// TIA Portal V19 export
DATA_BLOCK "Com_FromPolygonFiller"   // DB471
{ S7_Optimized_Access := 'TRUE' }
// stored: AutoNumber false, MemoryReserve 0
   VAR RETAIN
      CIP : Struct   // CIP Signals From Hassia
         LifeBit : Bool;   // Watchdog bit
         RequestCIPLye : Bool;   // Request Lye Only CIP
         RequestCIPLyeAcid : Bool;   // Request Lye + Acid CIP
         SpareBool_0_3 : Bool;
         SpareBool_0_4 : Bool;
         SpareBool_0_5 : Bool;
         SpareBool_0_6 : Bool;
         SpareBool_0_7 : Bool;
         CIPRunning : Bool;
         NoTimeStop : Bool;
         ReleaseCIPFeedPump : Bool;
         CipReturnPumpRunning : Bool;
         RequestPreRinse_1 : Bool;
         DrainMachine : Bool;
         RequestPreRinse_2 : Bool;
         RequestCaustic : Bool;
         RequestCausticRinse : Bool;   // Request Clear Rinse After Caustic
         RequestAcid : Bool;
         RequestAcidRinse : Bool;   // Request Clear Rinse After Acid
         MachineCleaned : Bool;
         SpareBool_2_4 : Bool;
         SpareBool_2_5 : Bool;
         SpareBool_2_6 : Bool;
         SpareBool_2_7 : Bool;
         SpareBool_3_0 : Bool;
         SpareBool_3_1 : Bool;
         SpareBool_3_2 : Bool;
         SpareBool_3_3 : Bool;
         SpareBool_3_4 : Bool;
         SpareBool_3_5 : Bool;
         SpareBool_3_6 : Bool;
         SpareBool_3_7 : Bool;
         Spacer : Array[0..11] of Word;
      END_STRUCT;
      SIP : Struct   // Sterilisation Signals from Hassia
         Request : Bool;
         Running : Bool;
         Sterile : Bool;   // Machine Sterile
         Spacer : Array[0..12] of Word;
      END_STRUCT;
      Production : Struct   // Production Signals from Hassia
         RequestFiller1 : Bool;
         StartProductPumpFiller1 : Bool;
         RequestFiller2 : Bool;
         StartProductPumpFiller2 : Bool;
         HopperLevelFiller1 : Int;
         HopperLevelFiller2 : Int;
         Spacer : Array[0..10] of Word;
      END_STRUCT;
   END_VAR
BEGIN
END_DATA_BLOCK
